INTERFACE I_Error EXTENDS __SYSTEM.IQueryInterface

METHOD PUBLIC Accept
VAR_INPUT
	Visitor : I_ErrorVisitor;
END_VAR
END_METHOD

PROPERTY PUBLIC Active : BOOL
GET
END_GET
END_PROPERTY

PROPERTY PUBLIC Message : T_MaxString
GET
END_GET
END_PROPERTY

PROPERTY PUBLIC Reason : T_MaxString
GET
END_GET
END_PROPERTY

END_INTERFACE

(* stored: Version 1.1.0.1, ProductVersion 3.1.4024.12
   Itf I_Error: Id {ac6f2e39-df03-0ea5-3235-056999a71a99}
   Method Accept: Id {b5a5ac7f-f823-064d-32bb-6a2242bbb63d}
   Property Active: Id {b3c89fa9-2658-0c39-24ec-48399945f1ef}
   Get Get: Id {55d61fc5-8c53-091d-15b8-d83ac1a9b91b}
   Property Message: Id {699dfe8b-6ccb-058e-3da7-73441f2ce52c}
   Get Get: Id {53371627-a92f-0249-3cb6-411a11b8dec0}
   Property Reason: Id {ace215d6-c0e0-0316-09e3-556a3e944761}
   Get Get: Id {5873fe10-6a68-00f4-0e9b-c7cf8a9cb704} *)
